(* IEC 61131-3 sources: CodesysTest/alpha/export/Device.dev/Plc Logic/Application/Programs, 2 files *)

(* ---- PRG_Bagger.pou.st ---- *)
(*#-#-#-#-#-#-#-#-#-#---Declaration---#-#-#-#-#-#-#-#-#-#-#-#-#*)

PROGRAM PRG_Bagger
VAR_INPUT

END_VAR
VAR_OUTPUT

END_VAR
VAR
    moabHead : FB_MOABHead_Electric;
    //angledHead : FB_20degHead();
    //pneuHead : FB_PneumaticHead();
    testEIPMotor : FB_AppliedMotionStepServoEIPBase();
    faultHandler : FB_FaultHandler();
	hmiInitiate : BOOL;
	msfMotorFaults : ARRAY[0..100] OF MotorCommFault;
	numberOfMSFFaults : UINT;
	msfCommFaultONS : R_TRIG();
	msfFaultListFull : BOOL;
	festoFaults : ARRAY[0..100] OF MotorCommFault;
	numberOfFestoFaults : UINT;
	festoCommFaultONS : R_TRIG();
	festoFaultListFull : BOOL;
	currentDateAndTime : GetTime();
	resetCommFaults : BOOL;
	i : INT;
	reverseFault : FB_HMIFault := (refFault := PRG_Bagger.moabHead.bagDelivery.reverseFault);
	faultActiveONS : FB_ONS;
END_VAR
(*#-#-#-#-#-#-#-#-#-#---Implementation---#-#-#-#-#-#-#-#-#-#-#-#-#*)

//    Program: PRG_Bagger
//    Description: This program glues together the whole machine and all of its components.
//
//    Created by: Ben Hess
//    Created Date: Tuesday, April 17, 2018

moabHead();
//pneuHead();
faultHandler();
hmiInitiate := HMIData.initiateCycle;
currentDateAndTime();
//msfCommFaultONS(CLK := MSFMotor.eState <> IoDrvEthernetIP.AdapterState.RUNNING);
HMIData.bagEdgePhotoeyeCovered := NOT iBagNotPresent;
oSoftStart := TRUE;

HMIData.airFilterClean();
HMIData.pressureBarGuideShaftGuides();
HMIData.driveRollerClean();
HMIData.printHeadClean();
//HMIData.pressureBarLeak(iExtended := iPressureBarExtended, iRetracted := iPressureBarRetracted, maximumStrokeTime := (TO_REAL(HMIData.passthroughSetting / 26.6)) + 0.3);
HMIData.loadPlateLeak(iExtended := iLoadPlateExtended, iRetracted := iLoadPlateRetracted, maximumStrokeTime := 0.4);
//HMIData.msfHorizontalMotorTemp(iDriveTemp := sealFlattenerHorizontalMotorInputs[4]);
//HMIData.bagDeliveryMotorTemp(iDriveTemp := bagDeliveryMotorInputs[4]);
//HMIData.passthroughMotorTemp(iDriveTemp := jawPasstrhoughMotorInputs[4]);

IF resetCommFaults THEN
	FOR i := 0 TO numberOfMSFFaults BY 1 DO
		msfMotorFaults[i].message := '';
		msfMotorFaults[i].timeOfFault := DT#1970-1-1-1:0:0;
	END_FOR
	numberOfMSFFaults := 0;
	msfFaultListFull := FALSE;
	resetCommFaults := FALSE;
END_IF

//HMIData.version := SVN_VERSION_INFO.VERSION;

HMIData.faultActive := GlobalObjects.CollectionOfActiveFaults.faultActive;
faultActiveONS(CLK := GlobalObjects.CollectionOfActiveFaults.faultActive);
IF faultActiveONS.OSR THEN
	moabHead.hmiLight.TurnOff();
END_IF

(* ---- PRG_MainProgram.pou.st ---- *)
(*#-#-#-#-#-#-#-#-#-#---Declaration---#-#-#-#-#-#-#-#-#-#-#-#-#*)

PROGRAM PRG_MainProgram
VAR
    incrementSolenoidCounter1 : R_TRIG();
    incrementSolenoidCounter2 : R_TRIG();
    incrementSolenoidFailedCounter2 : R_TRIG();
    GripperCycleCount : DINT; //Gripper Cycle Counter
    runPrinterPB : BOOL;
    cycleTimeMax : TIME;
    cycleTimeMaxDINT : DINT;
    ctfb : OSCAT_BASIC.CYCLE_TIME();
    profileThis :BOOL;
    solenoidState1 : SOLENOID_TEST_STATES;
    solenoidState2 : SOLENOID_TEST_STATES;
    getTimeTilPMMI : TimeLeftFB();
	displayPassthroughChangeDistance : REAL;
	displayPassthroughChangeDistance2 : REAL;
	checkSolenoid2ExtendTimer : TON := (PT := T#100MS);
	checkedSolenoid2Status : BOOL;
	firstScanDone : BOOL;
	printDeltaTimer : TON := (PT := T#5S);
	lastPrinterDelta : TIME;
	endPrintOSF : Standard.R_TRIG;
	//CSVWriter : FB_WriteToFile() := (xFilePath := 'C:/printerDelta.csv');
	stringToLog : STRING;
	testWrite : BOOL;
	hmiLight : FB_HMILight;
	versionInfo : VERSION;
	recipieManager : Recipe_Management.RecipeManCommands;
	recipeName : STRING;
	recResult : DWORD;
	testRead : BOOL;
	testCreate : BOOL;
	saveParametersTimer : Standard.TON := (PT := T#10M);
END_VAR(*#-#-#-#-#-#-#-#-#-#---Implementation---#-#-#-#-#-#-#-#-#-#-#-#-#*)

//    Program: Main (PLC_PRG)
//    Description: This program serves as a base for the MOAB Prototype
//    Created by: Ben Hess
//    Created Date: January 16th, 2018

printDeltaTimer(IN := oPrinterStartPrint);
saveParametersTimer(IN := NOT saveParametersTimer.Q);
IF saveParametersTimer.Q THEN
	recResult := recipieManager.GetRecipeNames('Recipes', ADR(recipeName),1,0);
	recResult := recipieManager.ReadAndSaveRecipe(RecipeDefinitionName := 'Recipes', RecipeName := recipeName);
	saveParametersTimer.IN := FALSE;
END_IF

IF testCreate THEN
// 	recResult := recipieManager.CreateRecipe(RecipeDefinitionName := 'Recipes', RecipeName := 'Automatic');
// 	recResult := recipieManager.ReadAndSaveRecipe(RecipeDefinitionName := 'Recipes', RecipeName := recipeName);
 	testCreate := FALSE;
	SaveValues();
END_IF

IF testRead THEN
// 	recResult := recipieManager.GetRecipeNames('Recipes', ADR(recipeName),1,0);
// 	recResult := recipieManager.LoadAndWriteRecipe(RecipeDefinitionName := 'Recipes', RecipeName := recipeName);
 	testRead := FALSE;
	RecallValues();
END_IF

//
// CSVWriter(
// 	xFilePath:= ,
// 	xText_Write:= ,
// 	xAppend_OverWrite:= TRUE,
// 	xAppend_Pos:= ,
// 	xWrite:= ,
// 	xRead:= ,
// 	xLine_No_To_Read:= ,
// 	xText_Read=> ,
// 	xDone=> );
// IF CSVWriter.xDone THEN
// 	CSVWriter.xWrite := FALSE;
// END_IF

ctfb(ct_max => cycleTimeMax);
cycleTimeMaxDINT := TIME_TO_DINT(cycleTimeMax);
profileThis := TIME_TO_DINT(ctfb.ct_last) >= 25;
// Run other programs
//PRG_PneumaticHead();
PRG_Bagger();
Faults();
versionInfo := GetVersion();
HMIData.version := Standard.CONCAT(TO_STRING(versionInfo.uiMajor),'.');
	BPLog.AppendToString(ADR(HMIData.version), CONCAT(TO_STRING(versionInfo.uiMinor),'.'));
	BPLog.AppendToString(ADR(HMIData.version), CONCAT(TO_STRING(versionInfo.uiServicePack),'.'));
	BPLog.AppendToString(ADR(HMIData.version), TO_STRING(versionInfo.uiPatch));
	BPLog.AppendToString(ADR(HMIData.version), TO_STRING(GetTextProperty("VersionPostfix")));
IF NOT firstScanDone THEN
	GlobalObjects.CollectionOfLoggable.RegisterAll(internalLogger := Globals.SystemLog);
	GlobalObjects.CollectionOfInitialzable.InitializeAll();
	firstScanDone := TRUE;
	// After first scan turn off flag set by StartDone system event
	Globals.firstScan := FALSE;
END_IF

// Start executing objects that implement IExecuteAutomatically
IF firstScanDone THEN
	GlobalObjects.CollectionOfExecutable.ExecuteAll();
	Globals.SystemLog();
END_IF

IF HMIData.ackAllFaults THEN
	GlobalObjects.CollectionOfActiveFaults.AckAll();
	HMIData.ackAllFaults := FALSE;
END_IF

getTimeTilPMMI(targetDate := DT#2018-10-14-8:0:0);

//First scan flag is set by task handler and reset in main routine here
IF Globals.firstScan THEN
    Globals.firstScan := FALSE;
END_IF

displayPassthroughChangeDistance := (UDINT_TO_REAL(Globals.passthroughChangeDistance) / 10);
displayPassthroughChangeDistance2 := (UDINT_TO_REAL(Globals.passthroughChangeDistance2) / 10.0);
